{attribute 'GeneratedUsingTerminal: EL3001-0000-0017'}
{attribute addProperty BoxType "EL3001-0000-0017"}
{attribute addProperty Id "StatusAT %I*Status_F2CE6D917ValueAT %I*INT2"}
{attribute addProperty CRC "1245267073"}
{attribute addProperty Size "9"}
TYPE AI_Standard_4A394481 :
STRUCT
	{attribute addProperty Name "Status"}
	Status AT %I* : Status_F2CE6D91;
	{attribute addProperty Name "Value"}
	Value AT %I* : INT;
END_STRUCT
END_TYPE

(* stored: Version 1.2.0.0, ProductVersion 3.1.4024.9
   DUT AI_Standard_4A394481: Id {5c5f76cb-63a5-46a0-892e-bb8d6e5c2a2d} *)
